// TIA Portal project "RobotFactores_Fluidez_Nsegundos" (V15.1)

(* hardware
DEVICE "ET 200SP station_1"  ET 200SP-Station
   slot 0: "Rack_0"  Rack  6ES5 710-8MAx1
   slot 1: "PLC Silo Pruebas"  CPU 1512SP-1 PN  6ES7 512-1DK01-0AB0  V2.5
   slot 2: "DI 16x24VDC ST_1"  DI 16x24VDC ST  6ES7 131-6BH01-0BA0  V0.0
      slot 1: "DI 16x24VDC ST_1"  DI 16x24VDC ST
   slot 3: "DQ 16x24VDC/0.5A ST_1"  DQ 16x24VDC/0.5A ST  6ES7 132-6BH01-0BA0  V0.0
      slot 1: "DQ 16x24VDC/0.5A ST_1"  DQ 16x24VDC/0.5A ST
   slot 4: "AI 4xU/I 2-wire ST_1"  AI 4xU/I 2-wire ST  6ES7 134-6HD00-0BA1  V1.1
      slot 1: "AI 4xU/I 2-wire ST_1"  AI 4xU/I 2-wire ST
   slot 5: "AQ 4xU/I ST_1"  AQ 4xU/I ST  6ES7 135-6HD00-0BA1  V1.1
      slot 1: "AQ 4xU/I ST_1"  AQ 4xU/I ST
   slot 6: "Siwarex de pesaje"  SIWAREX WP321  7MH4 138-6AA00-0BA0
      slot 1: "SIWAREX WP321_1"  SIWAREX WP321  7MH4 138-6AA00-0BA0
   slot 7: "Módulo servidor_1"  Server module  6ES7 193-6PA00-0AA0  V1.1
      slot 1: "Módulo servidor_1"  Server module
   slot 127: "BA 2xRJ45"  BA 2xRJ45  6ES7 193-6AR00-0AA0  V0.0
      slot 32769: "Port_1"  6ES7 193-6AR00-0AA0
      slot 32770: "Port_2"  6ES7 193-6AR00-0AA0
*)

// ===== PLC "PLC Silo Pruebas"  CPU 1512SP-1 PN =====
// protected blocks, not shown: "SIWAREX_WP321"

VAR_GLOBAL   // PLC tag table "Default tag table"
   "INPUT_boton_start_I-0-0" AT %I0.0 : Bool;   // Entrada física | botón del gabinete | normalmente abierto
   "INPUT_boton_stop_I-0-1" AT %I0.1 : Bool;   // Entrada física | botón del gabinete | normalmente cerrado
   "INPUT_sensorMariposa_cerrado_I-0-4" AT %I0.4 : Bool;   // Entrada física
   "INPUT_sensorMariposa_abierto_I-0-5" AT %I0.5 : Bool;   // Entrada física
   "OUTPUT_Hz_VFD_QW2" AT %QW2 : Word;   // Salida física | variador | 0-27648 = 0-60 Hz
   "OUTPUT_motor_vibrador_Q-0-1" AT %Q0.1 : Bool;   // Salida física | on/off
   "OUTPUT_motor_husillo_Q-0-0" AT %Q0.0 : Bool;   // Salida física | on/off
   "OUTPUT_valvula_mariposa_Q-0-5" AT %Q0.5 : Bool;   // Salida física | on/off
   "INPUT_Hz_lectura_VFD_IW-6" AT %IW6 : Int;   // Entrada física | variador | 0-27648 = 0-60 Hz
END_VAR

DATA_BLOCK "StatusRobot"   // DB5
{ S7_Optimized_Access := 'FALSE' }
VERSION : 0.1
   VAR
      motor_husillo : Bool;
      valvula_mariposa : Bool;
      sensor_mariposa_open : Bool;
      sensor_mariposa_close : Bool;
      vibradorEncendido : Bool;
      Hz_variador_actual : Word;
      Tiempo_ciclo : DWord;
      celda_carga : Int;
      setpoint_actual : Int;
   END_VAR
BEGIN
END_DATA_BLOCK

DATA_BLOCK "ListaOrdenes"   // DB14
{ S7_Optimized_Access := 'FALSE' }
VERSION : 0.1
   VAR
      Segundos : Array[0..9] of Int;
      Index_Lista : Int;
   END_VAR
BEGIN
END_DATA_BLOCK

DATA_BLOCK "Flags&Temps"   // DB18
{ S7_Optimized_Access := 'FALSE' }
VERSION : 0.1
   VAR
      SCADA_boton_Iniciar_ciclo : Bool;
      SCADA_boton_Terminar_ciclo : Bool;
      flag_leerEvento : Bool;
      flag_FIN_ciclo : Bool;
      vibrar : Bool;
      abrir_mariposa : Bool;
      motor_modo_manual : Bool;
      FirstScanBit : Bool;
      motor_husillo : Bool;
      siwarex_LifeBit : Bool;
      timerVibrar_In : Bool;
      timerVibrar_Out : Bool;
      timerHusillo_In : Bool;
      timerHusillo_Out : Bool;
      timerEstable_In : Bool;
      timerEstable_Out : Bool;
      timerAbrirMariposa_In : Bool;
      timerAbrirMariposa_Out : Bool;
      timerTiempoMuerto_In : Bool;
      timerTiempoMuerto_Out : Bool;
      End_TimerVibrar : Bool;
      End_TimerHusillo : Bool;
      End_TimerEstable : Bool;
      End_TimerMariposa : Bool;
      End_TimerTiempoMuerto : Bool;
      flag_tiempoMuertoON : Bool;
      flag_tiempoEstableON : Bool;
      flag_pushSTART : Bool;
      flag_pushSTOP : Bool;
      flag_pushSTART_SCADA : Bool;
      flag_pushSTOP_SCADA : Bool;
      SetPointTimeIN_vibrar : Time := T#1S;
      tiempoActual_timerVibrar : Time;
      SetPointTimeIN_husillo : Time;
      tiempoActual_timerHusillo : Time;
      SetPointTimeIN_estable : Time := T#6S;
      tiempoActual_timerEstable : Time;
      SetPointTimeIN_mariposa : Time := T#4S;
      tiempoActual_timerMariposa : Time;
      SetPointTimeIN_tiempoMuerto : Time := T#2S;
      tiempoActual_tiempoMuerto : Time;
      tiempoAcumulado_prev : DWord;
      tiempoEstable : Time;
      FrecuenciaOperacion : Int := 27648;
      out_Hz : Int;
      ESTADO : Int := 0;
      tiempo_timerActual : Time;
   END_VAR
BEGIN
END_DATA_BLOCK

// folder: System blocks/Program resources

DATA_BLOCK "IEC_Timer_pulsoMotor"   // DB6
{ S7_Optimized_Access := 'TRUE' }
AUTHOR : Simatic
FAMILY : IEC
NAME : IEC_TMR
VERSION : 1.0
// stored: InstanceOfName IEC_TIMER
"IEC_TIMER"
BEGIN
END_DATA_BLOCK

DATA_BLOCK "IEC_Timer_pulsoVibrador"   // DB15
{ S7_Optimized_Access := 'TRUE' }
AUTHOR : Simatic
FAMILY : IEC
NAME : IEC_TMR
VERSION : 1.0
// stored: InstanceOfName IEC_TIMER
"IEC_TIMER"
BEGIN
END_DATA_BLOCK

DATA_BLOCK "IEC_Timer_dead_for_read"   // DB16
{ S7_Optimized_Access := 'TRUE' }
AUTHOR : Simatic
FAMILY : IEC
NAME : IEC_TMR
VERSION : 1.0
// stored: InstanceOfName IEC_TIMER
"IEC_TIMER"
BEGIN
END_DATA_BLOCK

DATA_BLOCK "IEC_Timer_estable"   // DB17
{ S7_Optimized_Access := 'TRUE' }
AUTHOR : Simatic
FAMILY : IEC
NAME : IEC_TMR
VERSION : 1.0
// stored: InstanceOfName IEC_TIMER
"IEC_TIMER"
BEGIN
END_DATA_BLOCK

DATA_BLOCK "IEC_Timer_pulsoMariposa"   // DB19
{ S7_Optimized_Access := 'TRUE' }
AUTHOR : Simatic
FAMILY : IEC
NAME : IEC_TMR
VERSION : 1.0
// stored: InstanceOfName IEC_TIMER
"IEC_TIMER"
BEGIN
END_DATA_BLOCK

// folder: (top level)

FUNCTION "Deteccion_flancos" : Void   // FC1, SCL
TITLE = Flancos_deteccion
{ S7_Optimized_Access := 'TRUE' }
AUTHOR : Rafa
VERSION : 0.1
// Deteccion de flancos y control de pulsos
BEGIN
   //**** Detecta el flanco de bajada para detectar cuando acabo el timer
   "F_TRIG_DB_vibrador"(CLK := "Flags&Temps".timerVibrar_Out,
                        Q => "Flags&Temps".End_TimerVibrar);

   "F_TRIG_DB_husillo"(CLK := "Flags&Temps".timerHusillo_Out,
                       Q => "Flags&Temps".End_TimerHusillo);

   "F_TRIG_DB_estable"(CLK:= "Flags&Temps".timerEstable_Out,
                       Q=> "Flags&Temps".End_TimerEstable);

   "F_TRIG_DB_mariposa"(CLK := "Flags&Temps".timerAbrirMariposa_Out,
                        Q => "Flags&Temps".End_TimerMariposa);

   "F_TRIG_DB_tiempoMuerto"(CLK:= "Flags&Temps".timerTiempoMuerto_Out,
                            Q=> "Flags&Temps".End_TimerTiempoMuerto);

   "F_TRIG_DB_botonGabineteSTOP"(CLK:="INPUT_boton_stop_I-0-1",
                                 Q=>"Flags&Temps".flag_pushSTOP);

   "R_TRIG_DB_botonGabineteSTART"(CLK:="INPUT_boton_start_I-0-0",
                                  Q=>"Flags&Temps".flag_pushSTART);

   "R_TRIG_DB_IniciarCiclo"(CLK:="Flags&Temps".SCADA_boton_Iniciar_ciclo,
                            Q=> "Flags&Temps".flag_pushSTART_SCADA);

   "R_TRIG_DB_TerminarCiclo"(CLK:="Flags&Temps".SCADA_boton_Terminar_ciclo,
                             Q=>"Flags&Temps".flag_pushSTOP_SCADA);

   IF "Flags&Temps".ESTADO = 0 THEN
       "Flags&Temps".End_TimerTiempoMuerto := FALSE;
       "Flags&Temps".End_TimerVibrar := FALSE;
       "Flags&Temps".End_TimerHusillo := FALSE;
       "Flags&Temps".End_TimerEstable := FALSE;
       "Flags&Temps".End_TimerMariposa := FALSE;
   END_IF;

   //*** Baja flancos para que inicien timer
   IF "Flags&Temps".timerHusillo_In THEN
       "Flags&Temps".timerHusillo_In := FALSE;
   END_IF;
   IF "Flags&Temps".timerVibrar_In THEN
       "Flags&Temps".timerVibrar_In := FALSE;
   END_IF;
   IF "Flags&Temps".timerAbrirMariposa_In THEN
       "Flags&Temps".timerAbrirMariposa_In := FALSE;
   END_IF;
   IF "Flags&Temps".timerEstable_In THEN
       "Flags&Temps".timerEstable_In := FALSE;
   END_IF;
   IF "Flags&Temps".timerTiempoMuerto_In THEN
       "Flags&Temps".timerTiempoMuerto_In := FALSE;
   END_IF;
   IF "Flags&Temps".SCADA_boton_Terminar_ciclo THEN
       "Flags&Temps".SCADA_boton_Terminar_ciclo := FALSE;
   END_IF;
   IF "Flags&Temps".SCADA_boton_Iniciar_ciclo THEN
       "Flags&Temps".SCADA_boton_Iniciar_ciclo := FALSE;
   END_IF;
END_FUNCTION

FUNCTION "Asignaciones_finales" : Void   // FC2, SCL
TITLE = Asignaciones de variables
{ S7_Optimized_Access := 'TRUE' }
VERSION : 0.1
// Lo hace al final del main
BEGIN
   // Asignar valores - MOVE 

   "Flags&Temps".out_Hz := NORM_X_REAL(MIN := 0.0, MAX := 27648.0, VALUE := SCALE_X_REAL(MIN := 0.0, MAX := 60.0, VALUE := "INPUT_Hz_lectura_VFD_IW-6"));

   //"Hz VFD" := 13824;//  27648 = 60 hz  |  18432 = 40 hz  |  13824 = 30 hz  |  9216 = 20 hz
   "OUTPUT_Hz_VFD_QW2" := INT_TO_WORD("Flags&Temps".FrecuenciaOperacion);

   IF NOT "Flags&Temps".motor_modo_manual THEN
       "OUTPUT_motor_husillo_Q-0-0" := "Flags&Temps".motor_husillo;
   END_IF;

   "OUTPUT_motor_vibrador_Q-0-1" := "Flags&Temps".vibrar;
   "OUTPUT_valvula_mariposa_Q-0-5" := "Flags&Temps".abrir_mariposa;

   // Status
   "StatusRobot".valvula_mariposa := "OUTPUT_valvula_mariposa_Q-0-5";
   "StatusRobot".motor_husillo := "OUTPUT_motor_husillo_Q-0-0";
   "StatusRobot".Hz_variador_actual := INT_TO_WORD("Flags&Temps".out_Hz);


   CASE "Flags&Temps".ESTADO OF
       1: "Flags&Temps".tiempo_timerActual := "Flags&Temps".tiempoActual_tiempoMuerto;
       2: "Flags&Temps".tiempo_timerActual := "Flags&Temps".tiempoActual_timerVibrar;
       3: "Flags&Temps".tiempo_timerActual := "Flags&Temps".tiempoActual_timerHusillo;
       4: "Flags&Temps".tiempo_timerActual := "Flags&Temps".tiempoActual_timerEstable;
       5: "Flags&Temps".tiempo_timerActual := "Flags&Temps".tiempoActual_timerMariposa;
       ELSE
           "Flags&Temps".tiempo_timerActual := T#0S;
   END_CASE;

   "StatusRobot".Tiempo_ciclo := TIME_TO_DWORD("Flags&Temps".tiempo_timerActual) + "Flags&Temps".tiempoAcumulado_prev;
   "StatusRobot".sensor_mariposa_open := "INPUT_sensorMariposa_abierto_I-0-5";
   "StatusRobot".sensor_mariposa_close := "INPUT_sensorMariposa_cerrado_I-0-4";
   "StatusRobot".celda_carga := REAL_TO_INT("SIWAREX_WP321_DB".s_IO_DATA.PROCESS_VAL_1 * 1000);
   "StatusRobot".vibradorEncendido := "OUTPUT_motor_vibrador_Q-0-1";
END_FUNCTION

FUNCTION "Fin_dosificacion" : Void   // FC3, SCL
TITLE = Fin de dosificiación
{ S7_Optimized_Access := 'TRUE' }
VERSION : 0.1
// Al terminar el ciclo de dosificar
BEGIN
       "Flags&Temps".flag_leerEvento := FALSE;
       "Flags&Temps".flag_FIN_ciclo := TRUE;
       "Flags&Temps".ESTADO := 0;
       "Reiniciar_timers&values"();
END_FUNCTION

FUNCTION "Temporizadores" : Void   // FC4, SCL
TITLE = Timers
{ S7_Optimized_Access := 'TRUE' }
VERSION : 0.1
BEGIN
   //**** Timers

   "IEC_Timer_dead_for_read".TOF(IN:= "Flags&Temps".timerTiempoMuerto_In,
                                 PT:= "Flags&Temps".SetPointTimeIN_tiempoMuerto,
                                 Q => "Flags&Temps".timerTiempoMuerto_Out,
                                 ET => "Flags&Temps".tiempoActual_tiempoMuerto);

   "IEC_Timer_pulsoVibrador".TOF(IN := "Flags&Temps".timerVibrar_In,
                                 PT := "Flags&Temps".SetPointTimeIN_vibrar,
                                 Q => "Flags&Temps".timerVibrar_Out,
                                 ET => "Flags&Temps".tiempoActual_timerVibrar);

   "IEC_Timer_pulsoMotor".TOF(IN := "Flags&Temps".timerHusillo_In,
                              PT := "Flags&Temps".SetPointTimeIN_husillo,
                              Q => "Flags&Temps".timerHusillo_Out,
                              ET => "Flags&Temps".tiempoActual_timerHusillo);

   "IEC_Timer_estable".TOF(IN := "Flags&Temps".timerEstable_In,
                           PT := "Flags&Temps".SetPointTimeIN_estable,
                           Q => "Flags&Temps".timerEstable_Out,
                           ET => "Flags&Temps".tiempoActual_timerEstable);

   "IEC_Timer_pulsoMariposa".TOF(IN := "Flags&Temps".timerAbrirMariposa_In,
                                 PT := "Flags&Temps".SetPointTimeIN_mariposa,
                                 Q => "Flags&Temps".timerAbrirMariposa_Out,
                                 ET => "Flags&Temps".tiempoActual_timerMariposa);
END_FUNCTION

FUNCTION "Reiniciar_timers&values" : Void   // FC5, SCL
{ S7_Optimized_Access := 'TRUE' }
VERSION : 0.1
BEGIN
       // Reiniciar temporizadores
       RESET_TIMER("IEC_Timer_dead_for_read");
       RESET_TIMER("IEC_Timer_pulsoVibrador");
       RESET_TIMER("IEC_Timer_pulsoMotor");
       RESET_TIMER("IEC_Timer_estable");
       RESET_TIMER("IEC_Timer_pulsoMariposa");

       // Reiniciar Salidas del timer
       "Flags&Temps".timerTiempoMuerto_Out := FALSE;
       "Flags&Temps".timerVibrar_Out := FALSE;
       "Flags&Temps".timerHusillo_Out := FALSE;
       "Flags&Temps".timerEstable_Out := FALSE;
       "Flags&Temps".timerAbrirMariposa_Out := FALSE;

       // Reiniciar flags de visitado para cada ESTADO
       "Flags&Temps".flag_tiempoMuertoON := FALSE;
       "Flags&Temps".vibrar := FALSE;
       "Flags&Temps".motor_husillo := FALSE;
       "Flags&Temps".flag_tiempoEstableON := FALSE;
       "Flags&Temps".abrir_mariposa := FALSE;
END_FUNCTION

FUNCTION "PAROemergencia" : Void   // FC6, SCL
TITLE = Paro de Emergencia
{ S7_Optimized_Access := 'TRUE' }
VERSION : 0.1
// Definir los valores a tomar en un paro
BEGIN
   //la mariposa se queda en la posicion que se encuentra y se apagan los motores

   IF "INPUT_sensorMariposa_abierto_I-0-5" THEN
       "OUTPUT_valvula_mariposa_Q-0-5" := TRUE;
   ELSE
       "OUTPUT_valvula_mariposa_Q-0-5" := FALSE;
   END_IF;

   "OUTPUT_motor_husillo_Q-0-0" := FALSE;
   "OUTPUT_motor_vibrador_Q-0-1" := FALSE;
END_FUNCTION

FUNCTION "CMD_HANDLING" : Void   // FC30, SCL
{ S7_Optimized_Access := 'TRUE' }
VERSION : 0.1
   VAR_INPUT
      CMD_A : Int;
      CMD_B : Int;
      CMD3_In_Progress : Bool;
   END_VAR
   VAR_OUTPUT
      CMD3_TRIGGER : Bool;
   END_VAR
   VAR_IN_OUT
      CMD3_CODE : Int;
   END_VAR
BEGIN
   // Siwuarex

   IF (#CMD3_In_Progress=FALSE) THEN
     IF (#CMD_A<>0) THEN
       IF (#CMD_B<>0) THEN
         IF (#CMD3_CODE=#CMD_A) THEN #CMD3_CODE:=#CMD_B;
         ELSE #CMD3_CODE:=#CMD_A;
         END_IF;
       ELSE #CMD3_CODE:=#CMD_A;
       END_IF;
       #CMD3_TRIGGER:=TRUE;
     ELSIF (#CMD_B<>0) THEN #CMD3_CODE:=#CMD_B; #CMD3_TRIGGER:=TRUE;
     END_IF;
    END_IF;
END_FUNCTION

ORGANIZATION_BLOCK "Main"   // OB1, LAD, ProgramCycle
{ S7_Optimized_Access := 'TRUE' }
VERSION : 0.1
   VAR_INPUT
      Initial_Call : Bool;
      Remanence : Bool;
   END_VAR
BEGIN

REGION Network 1 (SCL): COMENTARIOS
   // Comentarios
   ///////////////////////////////////////////////////////////////////////
   ///////////////////////////////////////////////////
   //// 1Silo N_segundos N_dosificaciones
   ///////////////////////////////////////////////////////////////////////
   ///////////////////////////////////////////////////
   // Desde una BD en el ServerLocal, NodeRED actualiza la lista de dosificaciones.
   // Inicia la lectura de las variables del "status" del robot.
   // Cada una de las dosificaciones está representada por N segundos.
   // El programa espera un tiempo constante entre cada dosificiación.
   // Terminan las N dosificaciones y actualiza una bandera en NodeRED para terminar con la lectura de la BD en el ServerLocal
   ///////////////////////////////////////////////////////////////////////
   ///////////////////////////////////////////////////
   //
   //********************************************************************
   //
   // Version 1.0 Creado.      Lun17/08/20
   ////////// Problemas con el desfase del tiempo en LeerTiempo.
   // Version 1.1 TiempoCiclo := TOF.ET  +  TOF + Edge_Trigger
   ////////// Cambios en Lectura de tiempo de ejecucion + sin uso de bloques
   //
END_REGION

REGION Network 2: SIWAREX
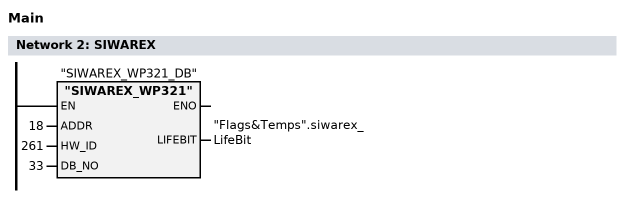
   RUNG wire#powerrail
      "SIWAREX_WP321_DB"(ADDR := 18, HW_ID := 261, DB_NO := 33, LIFEBIT => "Flags&Temps".siwarex_LifeBit)
   END_RUNG
   // the same network as SCL:
   "SIWAREX_WP321_DB"(ADDR := 18, HW_ID := 261, DB_NO := 33, LIFEBIT => "Flags&Temps".siwarex_LifeBit);   // "SIWAREX_WP321"
END_REGION

REGION Network 3 (SCL): PRINCIPAL
   // Importante: dejar Temporizadores() 
   "Temporizadores"();
   "Deteccion_flancos"();

   //**** Estados
   // 0: StandBy
   // 1: Tiempo muerto (Empieza a leer)    ESPERA
   // 2: Vibrar                            VIBRAR
   // 3: Prender motor husillo             HUSILLO
   // 4: Tiempo de estabilizacion          ESTABLE
   // 5: Abrir mariposa                    DESFOGUE
   // 6: Fin de 1 ciclo
   // 7: Fin de ejecución


   // 0: INICIAR CICLO
   IF "Flags&Temps".ESTADO = 0 AND ("Flags&Temps".flag_pushSTART_SCADA OR "Flags&Temps".flag_pushSTART)  THEN
       "Flags&Temps".SCADA_boton_Iniciar_ciclo := FALSE;
       "Flags&Temps".ESTADO := 1;
       "Flags&Temps".flag_leerEvento := TRUE;  // comienza a guardar en MSSQL_dbo.StatusRobot 
       "Flags&Temps".flag_FIN_ciclo := FALSE;
       "Flags&Temps".tiempoAcumulado_prev := 0;
       "ListaOrdenes".Index_Lista := 0;
       "OUTPUT_valvula_mariposa_Q-0-5" := FALSE;   // por si en el paro de emergencia quedó abierta
   END_IF;


   // 1: TIEMPO MUERTO
   IF "Flags&Temps".ESTADO = 1 AND NOT "Flags&Temps".flag_tiempoMuertoON THEN
       "Reiniciar_timers&values"();
       //Para avanzar si el tiempo es 0
       IF TIME_TO_DWORD("Flags&Temps".SetPointTimeIN_tiempoMuerto) = 0 THEN
           "Flags&Temps".ESTADO := 2;
       ELSE
           "Flags&Temps".timerTiempoMuerto_In := TRUE;       //inicia Timer
           "Flags&Temps".flag_tiempoMuertoON := TRUE;
       END_IF;
   END_IF;
   // Al terminar el timer de TiempoMuerto
   IF "Flags&Temps".End_TimerTiempoMuerto THEN
       "Flags&Temps".flag_tiempoMuertoON := FALSE;
       "Flags&Temps".ESTADO := 2;
       "Flags&Temps".tiempoAcumulado_prev := "Flags&Temps".tiempoAcumulado_prev + TIME_TO_DWORD("Flags&Temps".SetPointTimeIN_tiempoMuerto);
   END_IF;


   // 2: VIBRAR
   IF "Flags&Temps".ESTADO = 2 AND NOT "Flags&Temps".vibrar THEN
       //Para evitar vibrar si el tiempo es 0
       IF TIME_TO_DWORD("Flags&Temps".SetPointTimeIN_vibrar) = 0 THEN
           "Flags&Temps".ESTADO := 3;
       ELSE
           "Flags&Temps".timerVibrar_In := TRUE;       //inicia Timer
           "Flags&Temps".vibrar := TRUE;
       END_IF;
   END_IF;
   // Al terminar el timer de Vibrar
   IF "Flags&Temps".End_TimerVibrar THEN
       "Flags&Temps".vibrar := FALSE;
       "Flags&Temps".ESTADO := 3;
       "Flags&Temps".tiempoAcumulado_prev := "Flags&Temps".tiempoAcumulado_prev + TIME_TO_DWORD("Flags&Temps".SetPointTimeIN_vibrar);
   END_IF;


   // 3: HUSILLO
   IF "Flags&Temps".ESTADO = 3 AND NOT "Flags&Temps".motor_husillo THEN
       //Para terminar si el tiempo es 0
       IF "ListaOrdenes".Segundos["ListaOrdenes".Index_Lista] = 0 THEN
           "Flags&Temps".ESTADO := 6;
       ELSE
           // Asigna al SetPoint el valor siguiente de la lista de ordenes
           "StatusRobot".setpoint_actual := "ListaOrdenes".Segundos["ListaOrdenes".Index_Lista];
           "Flags&Temps".SetPointTimeIN_husillo := INT_TO_DINT("StatusRobot".setpoint_actual) * 1000;
           "Flags&Temps".timerHusillo_In := TRUE;             //inicia Timer
           "Flags&Temps".motor_husillo := TRUE;
       END_IF;
   END_IF;
   // Al terminar el timer del Husillo
   IF "Flags&Temps".End_TimerHusillo THEN
       "StatusRobot".setpoint_actual := 0;
       "ListaOrdenes".Index_Lista := "ListaOrdenes".Index_Lista + 1;
       "Flags&Temps".motor_husillo := FALSE;
       "Flags&Temps".ESTADO := 4;
       "Flags&Temps".tiempoAcumulado_prev := "Flags&Temps".tiempoAcumulado_prev + TIME_TO_DWORD("Flags&Temps".SetPointTimeIN_husillo);
   END_IF;


   // 4: ESTABILIZACIÓN
   IF "Flags&Temps".ESTADO = 4  AND NOT "Flags&Temps".flag_tiempoEstableON THEN
       //Para avanzar si el tiempo es 0
       IF TIME_TO_DWORD("Flags&Temps".SetPointTimeIN_estable) = 0 THEN
           "Flags&Temps".ESTADO := 5;
       ELSE
           "Flags&Temps".timerEstable_In := TRUE;             //inicia Timer
           "Flags&Temps".flag_tiempoEstableON := TRUE;
       END_IF;
   END_IF;
   // Al terminar el timer de Estabilización
   IF "Flags&Temps".End_TimerEstable THEN  
       "Flags&Temps".flag_tiempoEstableON := FALSE;
       "Flags&Temps".ESTADO := 5;
       "Flags&Temps".tiempoAcumulado_prev := "Flags&Temps".tiempoAcumulado_prev + TIME_TO_DWORD("Flags&Temps".SetPointTimeIN_estable);
   END_IF;


   // 5: MARIPOSA
   IF "Flags&Temps".ESTADO = 5 AND NOT "Flags&Temps".abrir_mariposa THEN
       //Para avanzar si el tiempo es 0
       IF TIME_TO_DWORD("Flags&Temps".SetPointTimeIN_mariposa) = 0 THEN
           "Flags&Temps".ESTADO := 6;
       ELSE
           "Flags&Temps".timerAbrirMariposa_In := TRUE;       //inicia Timer
           "Flags&Temps".abrir_mariposa := TRUE;
       END_IF;
   END_IF;
   // Al terminar el timer de Mariposa
   IF "Flags&Temps".End_TimerMariposa THEN
       "Flags&Temps".abrir_mariposa := FALSE;
       "Flags&Temps".ESTADO := 6;
       "Flags&Temps".tiempoAcumulado_prev := "Flags&Temps".tiempoAcumulado_prev + TIME_TO_DWORD("Flags&Temps".SetPointTimeIN_mariposa);
   END_IF;


   // 6: FIN CICLO
   IF "Flags&Temps".ESTADO = 6 THEN
       // Se acabo
       IF "ListaOrdenes".Segundos["ListaOrdenes".Index_Lista] = 0 THEN
           "Flags&Temps".ESTADO := 7;
       ELSE
           "Flags&Temps".ESTADO := 1;
       END_IF;
   END_IF;

    // Al terminar la ultima dosificacion o recibir un TERMINAR CICLO
   IF "Flags&Temps".ESTADO = 7 OR "Flags&Temps".flag_pushSTOP_SCADA OR "Flags&Temps".flag_pushSTOP  THEN
       "Fin_dosificacion"();
   END_IF;

   "Asignaciones_finales"();

   // normalmente cerrado
   IF NOT "INPUT_boton_stop_I-0-1" THEN
       "PAROemergencia"();
   END_IF;
END_REGION
END_ORGANIZATION_BLOCK

ORGANIZATION_BLOCK "Startup"   // OB100, SCL, Startup
TITLE = "Complete Restart"
{ S7_Optimized_Access := 'TRUE' }
VERSION : 0.1
   VAR_INPUT
      LostRetentive : Bool;   // True if retentive data are lost
      LostRTC : Bool;   // True if date and time are lost
   END_VAR
BEGIN
   // Actualiza para indicar al SCADA que actuilice
   "Flags&Temps".FirstScanBit := TRUE;
END_ORGANIZATION_BLOCK